// LS Electric XG5000 project: 과년66_1_2
// PLC NewPLC
// module base 0 slot 0: 입출력 모듈:XBC-DR20S (DC 24V 입력 12점, 릴레이 출력 8점)

PROGRAM NewProgram (task: 스캔 프로그램)

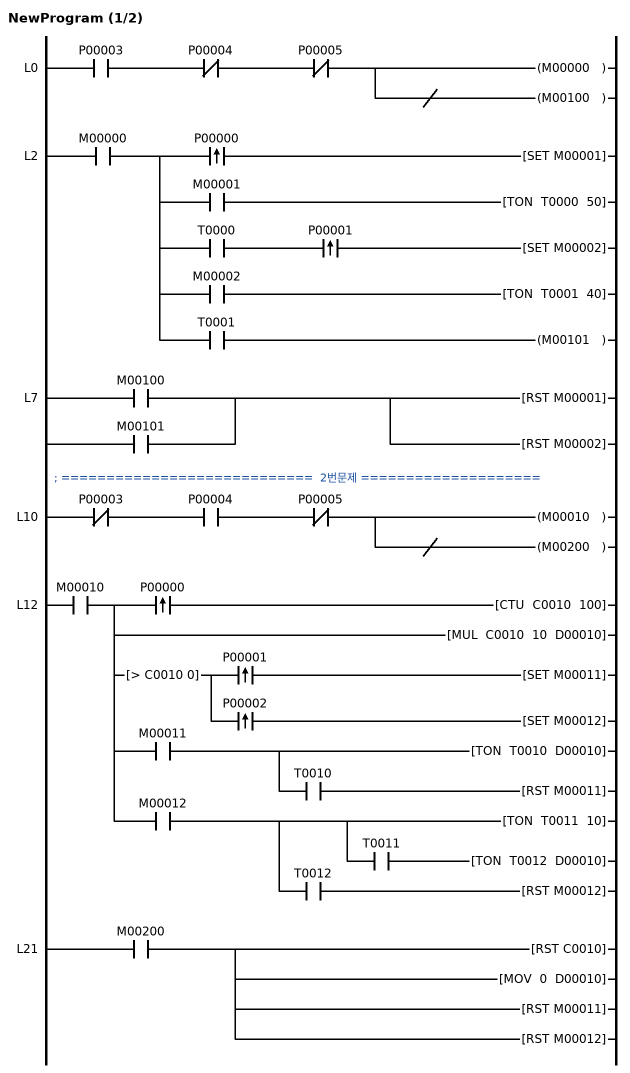
; L0
LOAD      P00003
AND NOT   P00004
AND NOT   P00005
OUT       M00000
NOT
OUT       M00100
; L2
LOAD      M00000
MPUSH
ANDP      P00000
SET       M00001
MLOAD
AND       M00001
TON       T0000 50
MLOAD
AND       T0000
ANDP      P00001
SET       M00002
MLOAD
AND       M00002
TON       T0001 40
MPOP
AND       T0001
OUT       M00101
; L7
LOAD      M00100
OR        M00101
RST       M00001
RST       M00002
// ============================  2번문제 ====================
; L10
LOAD NOT  P00003
AND       P00004
AND NOT   P00005
OUT       M00010
NOT
OUT       M00200
; L12
LOAD      M00010
MPUSH
ANDP      P00000
CTU       C0010 100
MLOAD
MUL       C0010 10 D00010
AND>      C0010 0
MPUSH
ANDP      P00001
SET       M00011
MPOP
ANDP      P00002
SET       M00012
MLOAD
AND       M00011
TON       T0010 D00010
AND       T0010
RST       M00011
MPOP
AND       M00012
TON       T0011 10
MPUSH
AND       T0011
TON       T0012 D00010
MPOP
AND       T0012
RST       M00012
; L21
LOAD      M00200
RST       C0010
MOV       0 D00010
RST       M00011
RST       M00012

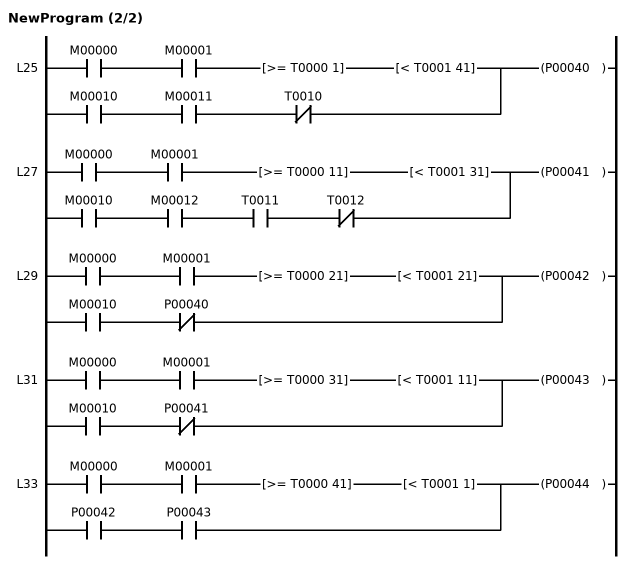
; L25
LOAD      M00000
AND       M00001
AND>=     T0000 1
AND<      T0001 41
LOAD      M00010
AND       M00011
AND NOT   T0010
OR LOAD
OUT       P00040
; L27
LOAD      M00000
AND       M00001
AND>=     T0000 11
AND<      T0001 31
LOAD      M00010
AND       M00012
AND       T0011
AND NOT   T0012
OR LOAD
OUT       P00041
; L29
LOAD      M00000
AND       M00001
AND>=     T0000 21
AND<      T0001 21
LOAD      M00010
AND NOT   P00040
OR LOAD
OUT       P00042
; L31
LOAD      M00000
AND       M00001
AND>=     T0000 31
AND<      T0001 11
LOAD      M00010
AND NOT   P00041
OR LOAD
OUT       P00043
; L33
LOAD      M00000
AND       M00001
AND>=     T0000 41
AND<      T0001 1
LOAD      P00042
AND       P00043
OR LOAD
OUT       P00044